// TIA Portal V17 export
// export: Created 2022-07-28T18:03:20.3807719Z, ExportSetting None, DisplayName Totally Integrated Automation Portal, DisplayVersion V17, DisplayName TIA Portal Openness, DisplayVersion V17, DisplayName TIA Portal Teamcenter Gateway, DisplayVersion V17, DisplayName TIA Portal Version Control Interface, DisplayVersion V17, DisplayName TIA Portal Test Suite Advanced, DisplayVersion V17, DisplayName SINAMICS Startdrive Advanced, DisplayVersion V17, DisplayName SINAMICS DCC, DisplayVersion V17, DisplayName SINAMICS Startdrive G130, G150, S120, S150, SINAMICS MV, S210, DisplayVersion V17, DisplayName SINAMICS Startdrive G110M, G120, G120C, G120D, G120P, G115D, DisplayVersion V17, DisplayName STEP 7 Professional, DisplayVersion V17, DisplayName SIMATIC Energy Suite, DisplayVersion V17, DisplayName STEP 7 CFC, DisplayVersion V17, DisplayName STEP 7 Safety, DisplayVersion V17, DisplayName WinCC Advanced / Unified PC, DisplayVersion V17, DisplayName SIMATIC Visualization Architect, DisplayVersion V17
TYPE "_PID_Cascad_Config"
   STRUCT
      "b" { ExternalAccessible := 'False'; ExternalVisible := 'False'; ExternalWritable := 'False'} : Struct   // bool parameters
         DirectMode { S7_SetPoint := 'True'} : Bool := true;   // 1 = Direct mode of PID choiced
         Enabled_P1 { S7_SetPoint := 'True'} : Bool := true;   // 1 = Pump 1 enabled for cascade
         Enabled_P2 { S7_SetPoint := 'True'} : Bool := true;   // 1 = Pump 2 enabled for cascade
         Enabled_P3 { S7_SetPoint := 'True'} : Bool := true;   // 1 = Pump 3 enabled for cascade
         bit_4 { S7_SetPoint := 'True'} : Bool;
         bit_5 { S7_SetPoint := 'True'} : Bool;
         bit_6 { S7_SetPoint := 'True'} : Bool;
         bit_7 { S7_SetPoint := 'True'} : Bool;
      END_STRUCT;
      r_SP_Auto_Value { S7_SetPoint := 'True'} : Real := 0.0;   // SP value for PID in auto mode, PU
      r_SP_Man_Value { S7_SetPoint := 'True'} : Real := 0.0;   // SP value for PID in auto mode, PU
      r_spP_part { S7_SetPoint := 'True'} : Real := 1.0;   // P part value
      r_spI_part { S7_SetPoint := 'True'} : Real := 20.0;   // I part value
      r_spD_part { S7_SetPoint := 'True'} : Real := 0.0;   // D part value
      r_FTC_Value { S7_SetPoint := 'True'} : Real := 0.0;   // Substitude value for forcely closed
      r_FTO_Value { S7_SetPoint := 'True'} : Real := 100.0;   // Substitude value for forcely opened
      r_Out_MaxValue { ExternalWritable := 'False'} : Real;   // Maximum value of output of PID
      r_Out_MinValue { ExternalWritable := 'False'} : Real;   // Minimum value of output of PID
      r_PV_MaxValue { ExternalWritable := 'False'} : Real;   // Maximum value of input of PID
      r_PV_MinValue { ExternalWritable := 'False'} : Real;   // Minimum value of input of PID
      r_spCascadeTime { S7_SetPoint := 'True'} : Real := 20.0;   // Time for on/off next stage of cascade
      r_spStabilizationTime : Real := 60.0;   // Time for stabilization detection, s
      r_ActSpeedSP_P1 { ExternalWritable := 'False'} : Real;   // Actual SP of speed, % of pump 1
      r_ActSpeedSP_P2 { ExternalWritable := 'False'} : Real := 0.0;   // Actual SP of speed, % of pump 2
      r_ActSpeedSP_P3 { ExternalWritable := 'False'} : Real := 0.0;   // Actual SP of speed, % of pump 3
      r_ActSpeedPV_P1 { ExternalWritable := 'False'} : Real;   // Actual PV of speed, % of pump 1
      r_ActSpeedPV_P2 { ExternalWritable := 'False'} : Real := 0.0;   // Actual PV of speed, % of pump 2
      r_ActSpeedPV_P3 { ExternalWritable := 'False'} : Real := 0.0;   // Actual PV of speed, % of pump 3
      r_Motohours_P1 { ExternalWritable := 'False'} : Real;   // Motohours of pump 1
      r_Motohours_P2 { ExternalWritable := 'False'} : Real := 0.0;   // Motohours of pump 2
      r_Motohours_P3 { ExternalWritable := 'False'} : Real := 0.0;   // Motohours of pump 3
      r_PV_ActValue { ExternalWritable := 'False'} : Real;   // Actual value of PV, PU
      r_Out_ActValue { ExternalWritable := 'False'} : Real;   // Actual value of output of PID, %
      r_QuanEnabled { ExternalWritable := 'False'} : Int;   // Quantity of enabled pumps
      i_Priority_P1 { S7_SetPoint := 'True'} : Int := 1;   // Priority of pump 1
      i_Priority_P2 { S7_SetPoint := 'True'} : Int := 2;   // Priority of pump 2
      i_Priority_P3 { S7_SetPoint := 'True'} : Int := 3;   // Priority of pump 3
      w_enableExternalErrors_16 { ExternalAccessible := 'False'; ExternalVisible := 'False'; ExternalWritable := 'False'; S7_SetPoint := 'True'} : Word := 16#FFFF;   // bit - 1 = enable
      b_bypassInterlocksForward_8 { ExternalAccessible := 'False'; ExternalVisible := 'False'; ExternalWritable := 'False'; S7_SetPoint := 'True'} : Byte := 16#FF;   // bit - 0 = Interlock Bypassed forward direction
      b_bypassInterlocksReverse_8 { ExternalAccessible := 'False'; ExternalVisible := 'False'; ExternalWritable := 'False'; S7_SetPoint := 'True'} : Byte := 16#FF;   // bit - 0 = Interlock Bypassed reverse direction
   END_STRUCT;
END_TYPE
